FUNCTION Convert_BOOL_TO_BOOL : BOOL
VAR_INPUT
	in : BOOL;
	out : REFERENCE TO BOOL;
END_VAR

out := in;
Convert_BOOL_TO_BOOL := TRUE;

END_FUNCTION

(* stored: Version 1.1.0.1, ProductVersion 3.1.4024.12
   POU Convert_BOOL_TO_BOOL: Id {0e932a57-8d49-4490-b6f3-0af122f0ca75}, SpecialFunc None *)
